// TIA Portal V20 export
// export: Created 2026-04-11T06:02:29.9153896Z, ExportSetting WithDefaults, DisplayName Totally Integrated Automation Portal, DisplayVersion V20, DisplayName TIA Portal Openness, DisplayVersion V20, DisplayName TIA Portal Version Control Interface, DisplayVersion V20, DisplayName STEP 7 Professional, DisplayVersion V20, DisplayName STEP 7 Safety, DisplayVersion V20, DisplayName WinCC Basic/Comfort/Advanced, DisplayVersion V20, DisplayName WinCC Unified, DisplayVersion V20
TYPE "udtError_SiwarexWP"
// stored: IsFailsafeCompliant false
   STRUCT
      CommandError { ExternalWritable := 'False'} : Bool;   // A command finished with an error
      AddressError { ExternalWritable := 'False'} : Bool;   // Incorrect hardware address
      RecordTransmissionFailed { ExternalWritable := 'False'} : Bool;   // Runtime error during transmission of data record
      ReadError { ExternalWritable := 'False'} : Bool;   // Reading of I/O data failed
      CommunicationLost { ExternalWritable := 'False'} : Bool;   // SiwarexWP module is not responding
      CommandSentAtStartup { ExternalWritable := 'False'} : Bool;   // Command was sent during startup
      DataRecordMismatch { ExternalWritable := 'False'} : Bool;   // Data record version does not match firmware
      InvalidCommand { ExternalWritable := 'False'} : Bool;   // An invalid command was sent to the module
      DataOperationError { ExternalWritable := 'False'} : Bool;   // Synchronous data operation error has occurred
      InternalFault { ExternalWritable := 'False'} : Bool;   // Module failed - replace the module
      LoadVoltageMissing { ExternalWritable := 'False'} : Bool;   // Low voltage - check supply voltage on module
      HardwareInterruptLost { ExternalWritable := 'False'} : Bool;   // Incorrect interrupt processing
      ModuleNotAvailable { ExternalWritable := 'False'} : Bool;   // Module is not ready for normal operation
      Undervoltage { ExternalWritable := 'False'} : Bool;   // Voltage drop to load cells is too large
      Overload { ExternalWritable := 'False'} : Bool;   // Scale overloaded
      Underload { ExternalWritable := 'False'} : Bool;   // Scale underloaded - check mechanical system
      ChecksumErrorInParameter { ExternalWritable := 'False'} : Bool;   // Incorrect parameters - reset to factory defaults
      ChecksumErrorInProgram { ExternalWritable := 'False'} : Bool;   // Incorrect module program - reset firmware or replace module
   END_STRUCT;
END_TYPE
